FUNCTION_BLOCK E_CHRON (* Event-driven Chronometer *)
  (* Standard: 61499-1; Classification: Event Processing; Function: Timing; Type: Elapsed time clock *)
  (* Version 0.1, 2002-01-29, JHC, Rockwell Automation, XML version *)
  (* Version 0.0, 1998-12-09, JHC, Rockwell Automation, SRC version *)
  (* Compiler header: package fb.rt.events; *)
  (* Compiler Java IBM VisualAge 3.0 *)
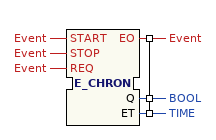
  EVENT_INPUT
    START; (* Start Timing *)
    STOP; (* Stop Timing *)
    REQ; (* Request readout *)
  END_EVENT
  EVENT_OUTPUT
    EO WITH Q, ET; (* Data Available *)
  END_EVENT
  VAR_OUTPUT
    Q : BOOL; (* 1=Running,0=Stopped *)
    ET : TIME; (* Time since last START up to STOP or REQ *)
  END_VAR
END_FUNCTION_BLOCK
